{attribute 'qualified_only'}
{attribute 'strict'}
{attribute 'to_string'}
TYPE E_HE_SATT_FilterStatus :
(
	DISABLED := 0,
    ENABLED
);
END_TYPE

(* stored: Version 1.1.0.1
   DUT E_HE_SATT_FilterStatus: Id {fb3ac64e-81fa-4550-b9d1-16ca1fbaf79e} *)
